{attribute 'qualified_only'}
{attribute 'strict'}
TYPE E_OpStep :
(
	IDLE := 0,
	START := 1,
	
	(* Pump Switchbox steps *)
	PSB_OPEN_GATE_VALVE,
	PSB_OPEN_PUMP_STATION_VALVES,
	PSB_ROUGH_CHAMBER,
	PSB_TURBO_CHAMBER,
	PSB_SWITCH_TO_ION_PUMP,
	PSB_CLOSE_GATE_VALVE,
	PSB_STOP_TURBO_PUMP,
	PSB_FINISH,
	
	(* Slow Pump switchbox steps *)
	SPSB_OPEN_GATE_VALVE,
	SPSB_OPEN_PUMP_STATION_VALVES,
	SPSB_ROUGH_CHAMBER,
	SPSB_OPEN_FORELINE_VALVE,
	SPSB_TURBO_CHAMBER,
	SPSB_SWITCH_TO_ION_PUMP,
	SPSB_CLOSE_VALVES,
	SPSB_STOP_TURBO_PUMP,
	SPSB_FINISH,
	
	(* Vent Switchbox steps *)
	VSB_CLOSE_GATE_VALVE,
	VSB_CLOSE_FORELINE_VALVE,
	VSB_TURN_OFF_PUMPS,
	VSB_CLOSE_ORING_VALVE,
	VSB_VENT,
	VSB_CLOSE_VENT,
	VSB_FINISH,
	
	(* Slow Vent Switchbox steps *)
	SVSB_CLOSE_GATE_VALVE,
	SVSB_CLOSE_FORELINE_VALVE,
	SVSB_TURN_OFF_PUMPS,
	SVSB_CLOSE_ORING_VALVE,
	SVSB_VENT,
	SVSB_SLOW_VENT,
	SVSB_CLOSE_VENT,
	SVSB_FINISH,
	
	(* Vent pump station *)
	VPS_VENT,
	VPS_CLOSE_VENT,
	VPS_FINISH,
	
	(* Pump Down Transport Tube *)
	POT_WAIT_PUMP_CART,
	POT_TURN_ON_PUMP,
	POT_FINISH,
	
	(* Vent Transport Tube *)
	VOT_VENT,
	VOT_WAIT_PC,
	VOT_FINISH,
	
	(* Open Transport Tube Gate Valve *)
	OTT_OPEN_VALVE
);
END_TYPE

(* stored: Version 1.1.0.1, ProductVersion 3.1.4022.17
   DUT E_OpStep: Id {ec262c74-2984-43a5-9b67-138f9035ebaf} *)
